Staubli VAL3: launchIdWD.pgx

program launchIdWD()
begin

  //if not existing launch moveid watchdog task
  if taskStatus("moveIdWatchdog")!=1
    taskKill("moveIdWatchdog")
    wait(taskStatus("moveIdWatchdog")==-1)
    taskCreate "moveIdWatchdog",10,moveIdWatchdog()
    wait(taskStatus("moveIdWatchdog")==1)
  endIf

end
